// TIA Portal V20 export
VAR_GLOBAL   // PLC tag table "LGR_Const_ToolType"
END_VAR
VAR_GLOBAL CONSTANT   // user constants
   TOOLTYPE_TBR : USInt := 1;   // TBR
   TOOLTYPE_PCR : USInt := 2;   // PCR
END_VAR
